Staubli VAL3: RosSimpleMsg.pjx

--- RosSimpleMsg.pjx ---
Parameters version=s7.7.2 stackSize=5000 millimeterUnit=true
Program file=start.pgx
Program file=stop.pgx
Data file=RosSimpleMsg.dtx
Type name=Prefix path=Disk://Prefix/Prefix.pjx
Type name=Header path=Disk://Header/Header.pjx
Type name=Body path=Disk://Body/Body.pjx

--- RosSimpleMsg.dtx ---
mdesc mNomSpeed
public Header header
  [0]
    num nMsgType
    num nCommType
    num nReplyCode
public Prefix prefix
  [0]
    num nLength
public Body body
  [0]
    num nData
